FUNCTION_BLOCK GR_plant
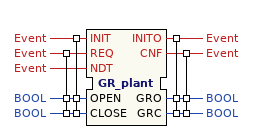
  EVENT_INPUT
    INIT WITH OPEN, CLOSE;
    REQ WITH OPEN, CLOSE;
    NDT;
  END_EVENT
  EVENT_OUTPUT
    INITO WITH GRO, GRC;
    CNF WITH GRO, GRC;
  END_EVENT
  VAR_INPUT
    OPEN : BOOL;
    CLOSE : BOOL;
  END_VAR
  VAR_OUTPUT
    GRO : BOOL;
    GRC : BOOL;
  END_VAR
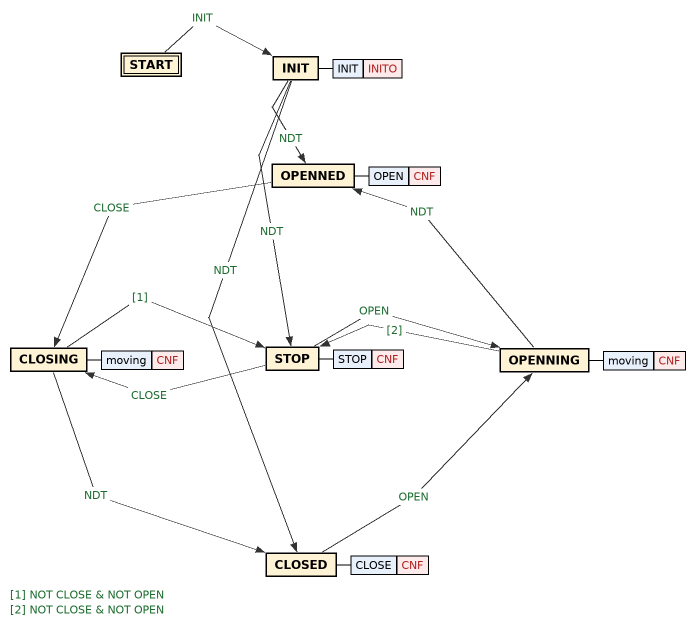
  EC_STATES
    START;
    INIT : INIT -> INITO;
    OPENNED : OPEN -> CNF;
    CLOSED : CLOSE -> CNF;
    OPENNING : moving -> CNF;
    CLOSING : moving -> CNF;
    STOP : STOP -> CNF;
  END_STATES
  EC_TRANSITIONS
    INIT TO OPENNED := NDT;
    CLOSING TO CLOSED := NDT;
    CLOSED TO OPENNING := OPEN;
    OPENNING TO OPENNED := NDT;
    OPENNED TO CLOSING := CLOSE;
    CLOSING TO STOP := NOT CLOSE & NOT OPEN;
    STOP TO OPENNING := OPEN;
    OPENNING TO STOP := NOT CLOSE & NOT OPEN;
    STOP TO CLOSING := CLOSE;
    INIT TO STOP := NDT;
    INIT TO CLOSED := NDT;
    START TO INIT := INIT;
  END_TRANSITIONS
  ALGORITHM INIT IN ST:
GRO := FALSE;
GRC := FALSE;
  END_ALGORITHM
  ALGORITHM OPEN IN ST:
GRO := TRUE;
GRC := FALSE;
  END_ALGORITHM
  ALGORITHM moving IN ST:
GRO := FALSE;
GRC := FALSE;
  END_ALGORITHM
  ALGORITHM CLOSE IN ST:
GRC := TRUE;
GRO := FALSE;
  END_ALGORITHM
  ALGORITHM STOP IN ST:
GRO := FALSE;
GRC := FALSE;
  END_ALGORITHM
END_FUNCTION_BLOCK
